FUNCTION F_RemoveInstancePathAndProjectNameFromTestInstancePath : Tc2_System.T_MaxString
VAR_INPUT
    TestInstancePath : Tc2_System.T_MaxString;
END_VAR
VAR
    CharacterPositionOfProjectName : INT;
    ProjectNameWithDot : Tc2_System.T_MaxString;
END_VAR

(* Add the '.' character to the project name for search *)
ProjectNameWithDot := Tc2_Standard.CONCAT(STR1 := TwinCAT_SystemInfoVarList._AppInfo.ProjectName, STR2 := '.');

(* Find the character position of the beginning of the first occurence of the project name *)
CharacterPositionOfProjectName := Tc2_Standard.FIND(STR1 := TestInstancePath, STR2 := ProjectNameWithDot);

IF CharacterPositionOfProjectName > 0 THEN
    TestInstancePath := Tc2_Standard.DELETE(STR := TestInstancePath,
                                            LEN := CharacterPositionOfProjectName-1 + Tc2_Standard.LEN(ProjectNameWithDot),
                                            POS := 1);
END_IF

(* Check if the project name happens to be the same as namespace, and in that case, remove that as well *)
CharacterPositionOfProjectName := Tc2_Standard.FIND(STR1 := TestInstancePath,
                                                    STR2 := ProjectNameWithDot);

IF CharacterPositionOfProjectName > 0 THEN
    TestInstancePath := Tc2_Standard.DELETE(STR := TestInstancePath,
                                            LEN := CharacterPositionOfProjectName - 1 + 
                                                Tc2_Standard.LEN(STR := ProjectNameWithDot),
                                            POS := 1);
END_IF

F_RemoveInstancePathAndProjectNameFromTestInstancePath := TestInstancePath;

END_FUNCTION

(* stored: Version 1.1.0.1, ProductVersion 3.1.4022.18
   POU F_RemoveInstancePathAndProjectNameFromTestInstancePath: Id {7816860e-5623-4ff0-b466-902e340371e3}, SpecialFunc None *)
